(* Logix 5000 project; controller Dobot_V1PLC 5069-L306ERM rev 33.11; software revision 33.00 *)

TASK MainTask (continuous, watchdog 500 ms) : MainProgram

MODULES
   Local : 5069-L306ERM (5069 0, rev 33.11)
       : vendor 1 type 7 code 391 (5069 1, rev 2.1, StandardDataDriven RPI 5 ms)
       : 5069-OB16 (5069 2, rev 2.1, StandardDataDriven RPI 5 ms)
END_MODULES

TYPE Sort_Array :   // This UDT will store values for a sorting method to use in order
STRUCT
   First_Color : STRING;
   Second_Color : STRING;
   Third_Color : STRING;
   Fourth_Color : STRING;
END_STRUCT
END_TYPE

ADD_ON_INSTRUCTION SS_AOI   (* revision 1.0 *)
// starting and stopping the conveyor and the dobot
VAR_INPUT
   Sys_On : BOOL; {required}
END_VAR
VAR_OUTPUT
   Run : BOOL; {access Read Only, required}
END_VAR
VAR_IN_OUT
   PRE_TMR : DINT; {required}
END_VAR
VAR_OUTPUT
   ACC_TMR : DINT; {access Read Only, visible}
END_VAR
VAR_IN_OUT
   Off : BOOL; {required}
END_VAR
VAR
   Delay : BOOL; {access None}
   Delay_TMR : TIMER; {access None}
END_VAR

ROUTINE Logic   (* ladder *)
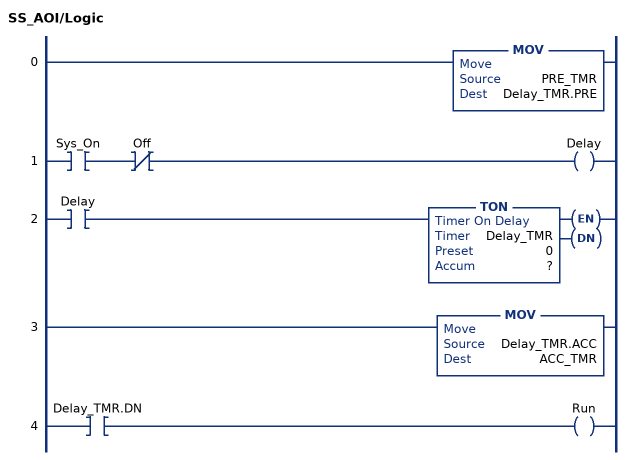
   0: MOV(PRE_TMR,Delay_TMR.PRE);
   1: XIC(Sys_On)XIO(Off)OTE(Delay);
   2: XIC(Delay)TON(Delay_TMR,?,?);
   3: MOV(Delay_TMR.ACC,ACC_TMR);
   4: XIC(Delay_TMR.DN)OTE(Run);
END_ROUTINE
END_ADD_ON_INSTRUCTION

VAR_GLOBAL   (* controller tags *)
   Color_STR : Sort_Array := (First_Color := 'g', Second_Color := 'r', Third_Color := 'r', Fourth_Color := 'g');
END_VAR

PROGRAM MainProgram   (* main routine MainRoutine *)
VAR
   All : BOOL := 1;
   Array_S : BOOL;
   Array_Sort : BOOL;
   Block_Count : DINT;
   Block_Detected : BOOL := 1;
   Blue : BOOL;
   Color : SINT := 3;
   Conv_Run : BOOL;
   Conv_Speed : DINT := 24;
   Current_Color : STRING := 'Yellow';
   Current_Sort : STRING := 'Random Sort';
   ESTOP : BOOL;
   Green : BOOL;
   HMI_String1 : STRING := 'G';
   HMI_String2 : STRING := 'R';
   HMI_String3 : STRING := 'R';
   HMI_String4 : STRING := 'G';
   HMI_String5 : STRING := 'B';
   Manual : BOOL;
   Manual_Sort : BOOL;
   Maxed_Out : BOOL;
   Random : BOOL := 1;
   Random_Sort : BOOL;
   Red : BOOL;
   Reset : BOOL;
   Reset_Count : BOOL;
   Same : BOOL;
   Same_Sort : BOOL;
   SL_SPD : DINT := 24;
   Sorting : STRING[5] := ([0] := 'G', [1] := 'R', [2] := 'R', [3] := 'G', [4] := 'B');
   Start : BOOL;
   Stop : BOOL;
   Suction_Run : BOOL;
   System_off : BOOL;
   System_Running : BOOL := 1;
   Yellow : BOOL;
END_VAR

ROUTINE Color_Sort_Selection   (* ladder *)
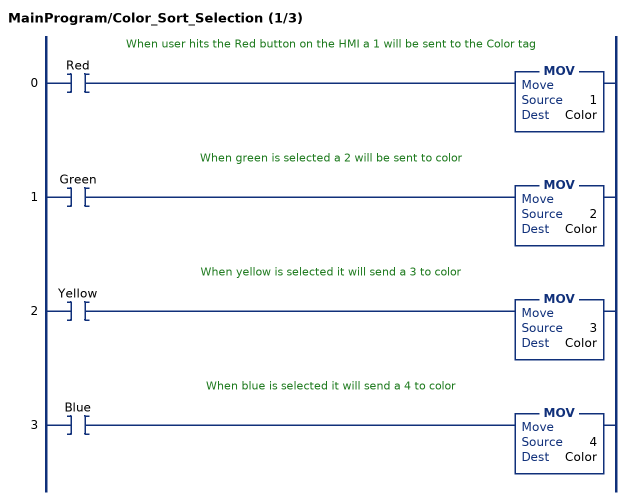
   // When user hits the Red button on the HMI a 1 will be sent to the Color tag
   0: XIC(Red)MOV(1,Color);
   // When green is selected a 2 will be sent to color
   1: XIC(Green)MOV(2,Color);
   // When yellow is selected it will send a 3 to color
   2: XIC(Yellow)MOV(3,Color);
   // When blue is selected it will send a 4 to color
   3: XIC(Blue)MOV(4,Color);
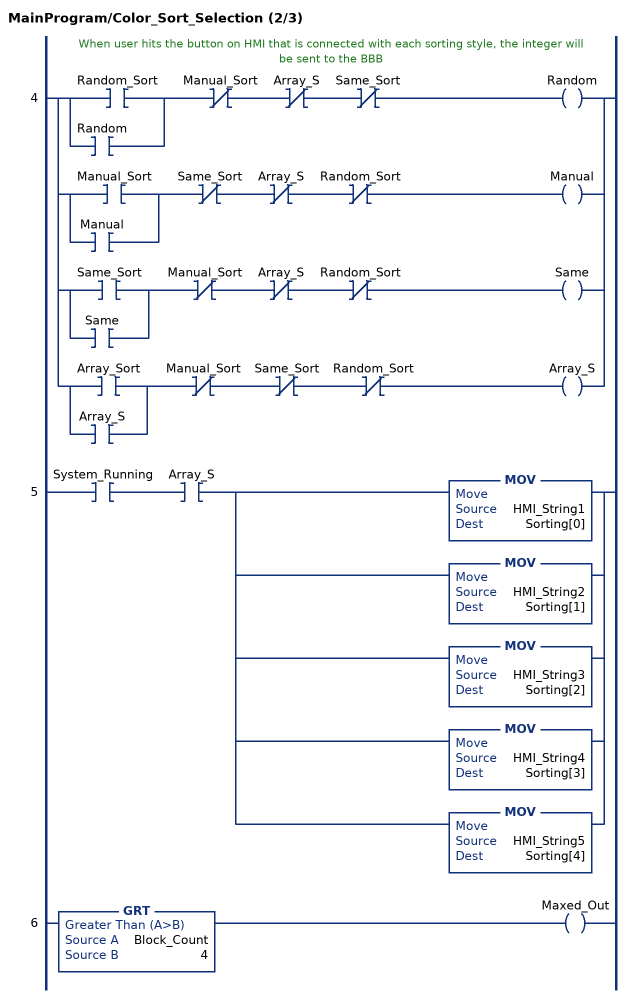
   // When user hits the button on HMI that is connected with each sorting style, the integer will be sent to the BBB
   4: [[XIC(Random_Sort) ,XIC(Random) ] XIO(Manual_Sort) XIO(Array_S) XIO(Same_Sort) OTE(Random) ,[XIC(Manual_Sort) ,XIC(Manual) ] XIO(Same_Sort) XIO(Array_S) XIO(Random_Sort) OTE(Manual) ,[XIC(Same_Sort) ,XIC(Same) ] XIO(Manual_Sort) XIO(Array_S) XIO(Random_Sort) OTE(Same) ,[XIC(Array_Sort) ,XIC(Array_S) ] XIO(Manual_Sort) XIO(Same_Sort) XIO(Random_Sort) OTE(Array_S) ];
   5: XIC(System_Running)XIC(Array_S)[MOV(HMI_String1,Sorting[0]) ,MOV(HMI_String2,Sorting[1]) ,MOV(HMI_String3,Sorting[2]) ,MOV(HMI_String4,Sorting[3]) ,MOV(HMI_String5,Sorting[4]) ];
   6: GRT(Block_Count,4)OTE(Maxed_Out);
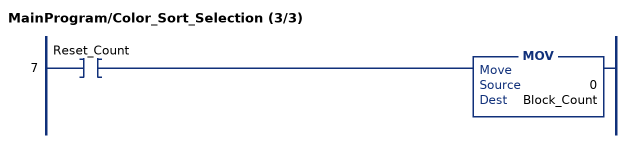
   7: XIC(Reset_Count)MOV(0,Block_Count);
END_ROUTINE

ROUTINE Main_Logic   (* ladder *)
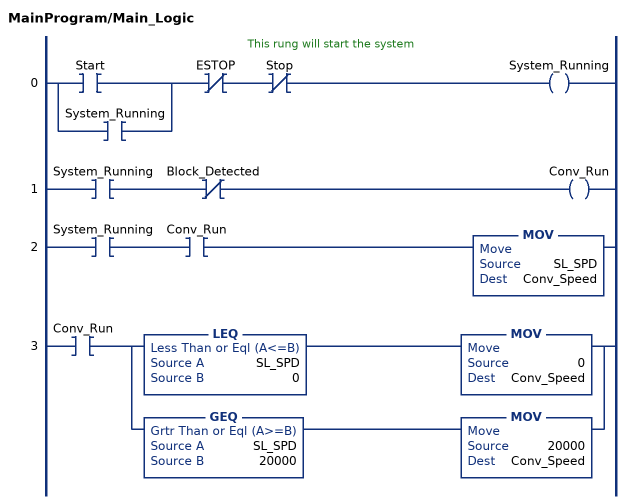
   // This rung will start the system
   0: [XIC(Start) ,XIC(System_Running) ]XIO(ESTOP)XIO(Stop)OTE(System_Running);
   1: XIC(System_Running)XIO(Block_Detected)OTE(Conv_Run);
   2: XIC(System_Running)XIC(Conv_Run)MOV(SL_SPD,Conv_Speed);
   3: XIC(Conv_Run)[LEQ(SL_SPD,0) MOV(0,Conv_Speed) ,GEQ(SL_SPD,20000) MOV(20000,Conv_Speed) ];
END_ROUTINE

ROUTINE MainRoutine   (* ladder *)
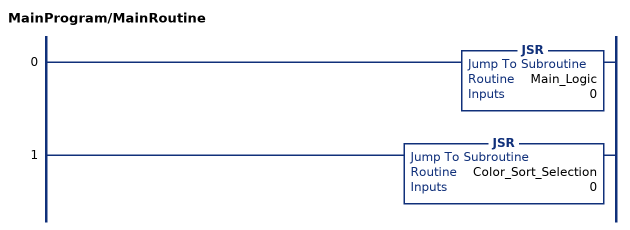
   0: JSR(Main_Logic,0);
   1: JSR(Color_Sort_Selection,0);
END_ROUTINE
END_PROGRAM
